FUNCTION_BLOCK CMP_OC_W10

VAR_INPUT
	BOOL_INTERLOCK : BOOL; (*INTERLOCK*)
	WORD_1: WORD;		(*WORD 1*)
	WORD_2: WORD;		(*WORD 2*)
	WORD_3: WORD;		(*WORD 3*)
	WORD_4: WORD;		(*WORD 4*)
	WORD_5: WORD;		(*WORD 5*)
	WORD_6: WORD;		(*WORD 6*)
	WORD_7: WORD;		(*WORD 7*)
	WORD_8: WORD;		(*WORD 8*)
	WORD_9: WORD;		(*WORD 9*)
	WORD_10: WORD;	(*WORD 10*)
END_VAR


VAR_OUTPUT
	BZ_OUTPUT_BOOL : BOOL;
END_VAR


VAR
	OUT_1: BOOL;
	OUT_2: BOOL;
	OUT_3: BOOL;
	OUT_4: BOOL;
	OUT_5: BOOL;
	OUT_6: BOOL;
	OUT_7: BOOL;
	OUT_8: BOOL;
	OUT_9: BOOL;
	OUT_10: BOOL;

END_VAR

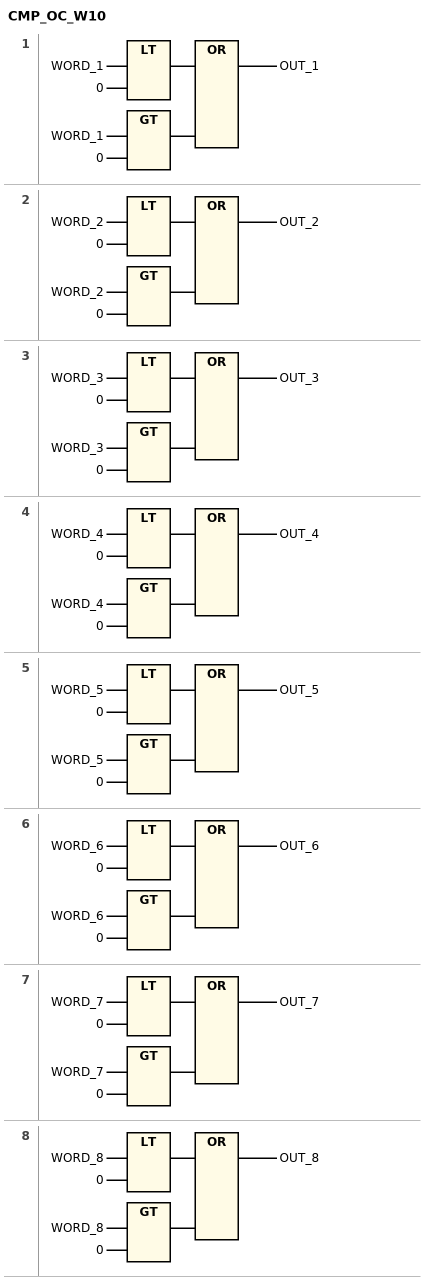
// NETWORK 1
OUT_1 := WORD_1 < 0 OR WORD_1 > 0;

// NETWORK 2
OUT_2 := WORD_2 < 0 OR WORD_2 > 0;

// NETWORK 3
OUT_3 := WORD_3 < 0 OR WORD_3 > 0;

// NETWORK 4
OUT_4 := WORD_4 < 0 OR WORD_4 > 0;

// NETWORK 5
OUT_5 := WORD_5 < 0 OR WORD_5 > 0;

// NETWORK 6
OUT_6 := WORD_6 < 0 OR WORD_6 > 0;

// NETWORK 7
OUT_7 := WORD_7 < 0 OR WORD_7 > 0;

// NETWORK 8
OUT_8 := WORD_8 < 0 OR WORD_8 > 0;

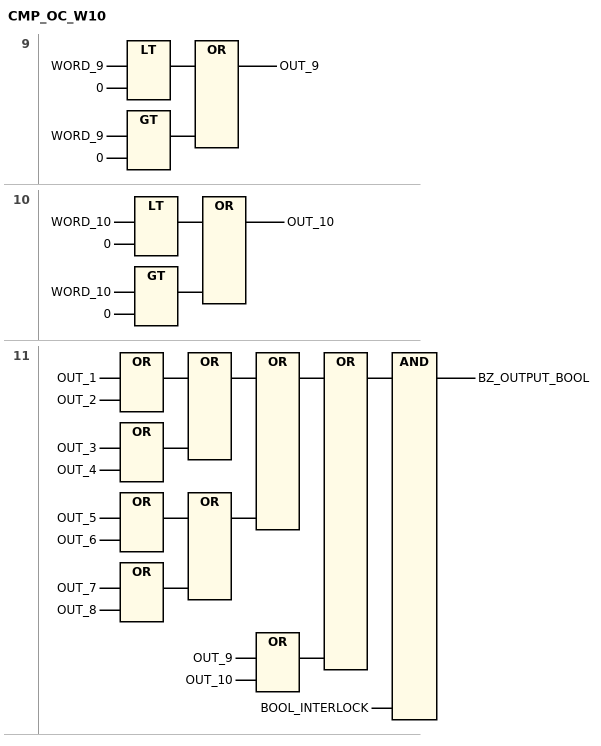
// NETWORK 9
OUT_9 := WORD_9 < 0 OR WORD_9 > 0;

// NETWORK 10
OUT_10 := WORD_10 < 0 OR WORD_10 > 0;

// NETWORK 11
BZ_OUTPUT_BOOL := ((((OUT_1 OR OUT_2) OR (OUT_3 OR OUT_4)) OR ((OUT_5 OR OUT_6) OR (OUT_7 OR OUT_8))) OR (OUT_9 OR OUT_10)) AND BOOL_INTERLOCK;

END_FUNCTION_BLOCK

(* stored: Version 1.1.0.1, ProductVersion 3.1.4024.12
   POU CMP_OC_W10: Id {22813178-1a11-4aee-9c4f-205c8300d026}, SpecialFunc None *)
